FUNCTION_BLOCK Room_State_Idle EXTENDS Room_State
VAR_INPUT
END_VAR
VAR_OUTPUT
END_VAR
VAR
END_VAR

METHOD OnEntry
_ctx.io.bOpenValves := FALSE;

_ctx.priv.bActive := FALSE;
_ctx.priv.bReady := FALSE;

_ctx.hmi.sStatusText := 'Heating ON: Idle';
_ctx.hmi.nStatusColor := COL.BLACK.Raw;

_ctx.hmi.bHideReset := FALSE;
END_METHOD

METHOD OnExecute
IF _ctx.hmi.bDisable THEN
	_ctx.state.iMgr.Request(_ctx.state.iDisable);
END_IF
END_METHOD

END_FUNCTION_BLOCK

(* stored: Version 1.1.0.1
   POU Room_State_Idle: Id {4c766015-91cf-477b-985f-581e4af963c5}, SpecialFunc None
   Method OnEntry: Id {d4b48581-1a4d-4829-a23f-cfc37a8808cd}
   Method OnExecute: Id {1f6e34fe-0771-4959-934b-53cc7be7116b} *)
